# EPICS autosave request: iocBoot/iocsrsDS345/auto_positions.req
file srsDS345_settings.req P=$(P)
